(* Logix 5000 project; controller AdvManLab vendor 1 type 14 code 158 rev 28.12; software revision 28.01; part 2 of 13 *)
(* tags used below, declared in another part *)
   Inp : BOOL;   // Alarm Condition Input 1=Alarm
   Inp_Reset : BOOL;   // 1=Reset Alarm requiring reset
   Cfg_Exists : BOOL;   // 1=Alarm configured to exist, 0=Does not exist, don't scan
   Cfg_ResetReqd : BOOL;   // 1=Latched Alarm, a Reset is required to clear this Alarm
   Cfg_AckReqd : BOOL;   // 1=Acknowledge required for this Alarm
   Cfg_AllowShelve : BOOL;   // 1=Allow Operator to Shelve this Alarm
   Cfg_AllowDisable : BOOL;   // 1=Allow Maintenance to Disable this Alarm
   Cfg_PCmdClear : BOOL;   // 1=Clear Program Commands on receipt 0=Leave Set
   Cfg_Severity : INT;   // Alarm Severity: 1..250=Low, 251..500=Medium, 501..750=High, 751..1000=Urgent
   Cfg_AlmMinOnT : DINT;   // Minimum time Alm output stays on (sec)
   Cfg_MaxShelfT : INT;   // Auto unshelve after shelved this long (1..32767 minutes)
   PCfg_AllowExist : BOOL;   // 1=Alarm can be configured to exist, 0=other configs make alarm meaningless
   PCmd_Reset : BOOL;   // Program Command to Reset latched alarm
   PCmd_Ack : BOOL;   // Program Command to Acknowledge alarm
   PCmd_Suppress : BOOL;   // Program Command to Suppress by Design (inhibits new alarm)
   PCmd_Unsuppress : BOOL;   // Program Command to Unsuppress (allows new alarm)
   PCmd_Unshelve : BOOL;   // Program Command to Unshelve (e.g., on shift change)
   OCmd_Reset : BOOL;   // Operator Command to Reset latched alarm
   OCmd_Ack : BOOL;   // Operator Command to Acknowledge alarm
   OCmd_Shelve : BOOL;   // Operator Command to Shelve Alarm (inhibits new alarm)
   OCmd_Unshelve : BOOL;   // Operator Command to Unshelve alarm (allows new alarm)
   MCmd_Disable : BOOL;   // Maintenance Command to Disable alarm (inhibits new alarm)
   MCmd_Enable : BOOL;   // Maintenance Command to Enable alarm (allows new alarm)
   MCmd_Test : BOOL;   // Maintenance Command to Test alarm (issued for minimum alarm time)
   Val_Notify : SINT;   // Current Alarm Severity and Acknowledgement (enumeration)
   Val_MinToUnshelve : DINT;   // Number of minutes until this alarm unshelves itself (mmm:ss)
   Val_SecToUnshelve : DINT;   // Number of Seconds until this alarm unshelves itself (mmm:ss)
   Alm : ALIAS FOR Com_AE.0;   // Alarm output 1=In Alarm
   Ack : ALIAS FOR Com_AE.1;   // Alarm acknowledged status: 1=Ack rcvd
   Shelved : ALIAS FOR Com_AE.3;   // 1=Alarm has been Shelved by Operator (inhibits new alarm)
   Suppressed : ALIAS FOR Com_AE.6;   // 1=Alarm has been Suppressed by Program (inhibits new alarm)
   Disabled : ALIAS FOR Com_AE.9;   // 1=Alarm has been Disabled by Maintanance (inhibits new alarm)
   Sts_AlmInh : BOOL;   // 1=Alarm has been suppressed, shelved or disabled, display "I" icon
   Sts_Err : BOOL;   // 1=Error in Config: see detail Err_ bits for reason
   Err_Timer : BOOL;   // 1=Error in Config: Alarm Min On Time, Shelf Time (use 0 to 2147483)
   Err_Severity : BOOL;   // 1=Error in Config: Invalid Severity (use 1 to 4)
   Rdy_Reset : BOOL;   // Ready to receive OCmd_Reset (enables button)
   Rdy_Ack : BOOL;   // Ready to receive OCmd_Ack (enables button)
   Rdy_Shelve : BOOL;   // Ready to receive OCmd_Shelve (enables button)
   Rdy_Unshelve : BOOL;   // Ready to receive OCmd_Unshelve (enables button)
   Rdy_Disable : BOOL;   // Ready to receive MCmd_Disable (enables button)
   Rdy_Enable : BOOL;   // Ready to receive MCmd_Enable (enables button)
   Rdy_Test : BOOL;   // Ready to receive MCmd_Test (enables button)
   P_Alarm : BOOL;   // Unique Parameter Name for auto - discovery
   Wrk_Alm : BOOL;   // Internal Alarm Status
   Wrk_Suppressed : BOOL;   // Internal Alarm Suppressed Status
   Wrk_AlmMinOnT : TIMER;   // Alarm output minimum ON time to be seen by alarm server
   Wrk_AutoAckT : TIMER;   // Time to clear Ack bit when Ack not required
   Wrk_ShelfT : TIMER;   // Time to auto Unshelve a Shelved Alarm
   Com_AE : INT;   // Communication with HMI / Alarm/Event Server (see bit descriptions)
   Cfg_Tag : STRING_20;   // Alarm Tag Text (e.g., "LAHH-101")
   Cfg_Cond : STRING_20;   // Alarm Condition Text (e.g., "High-High PV")
   Wrk_SecToUnshelve : DINT;   // Number of seconds until this alarm unshelves itself
   Inf_Lib : STRING_12;   // Display Library for Faceplate call-up
   Inf_Type : STRING_16;   // Must contain AOI name, used for HMI and Information S/W
(* P_Alarm, continued *)

ROUTINE EnableInFalse   (* ladder *)
// Perform Alarm processing, but Invert Alarm Input ("Inp") for use on LD rung (EnableIn False)
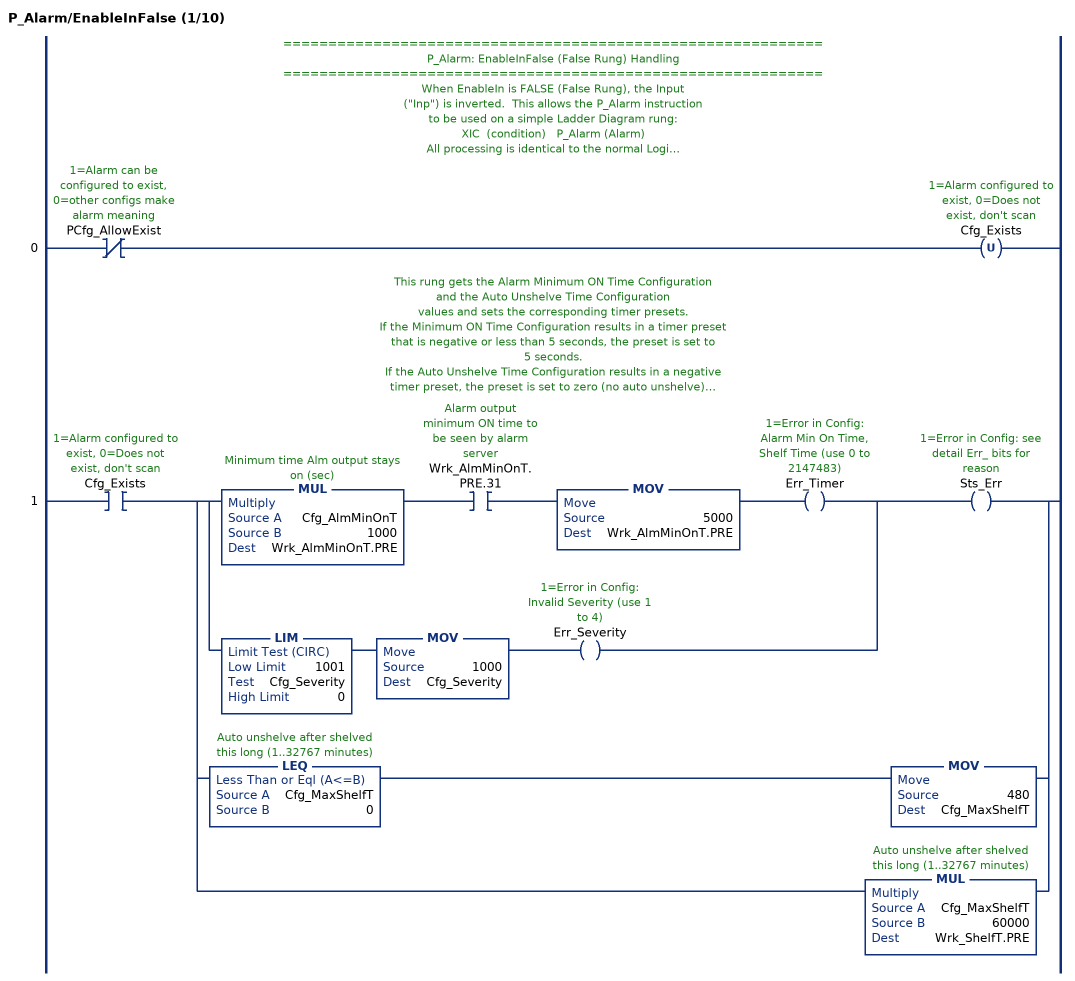
   // ============================================================
   // P_Alarm: EnableInFalse (False Rung) Handling
   // ============================================================
   // When EnableIn is FALSE (False Rung), the Input
   // ("Inp") is inverted.  This allows the P_Alarm instruction
   // to be used on a simple Ladder Diagram rung:
   // XIC  (condition)   P_Alarm (Alarm)
   // All processing is identical to the normal Logic
   // routine, except references to Inp are inverted!
   // ============================================================
   // CONFIGURATION
   // ============================================================
   // In the object containing this alarm, other configuration (such as not having
   // any limit switches) may make this particular alarm meaningless.
   // The Program Configuration "Allow Exist" is used to hide this alarm
   // on the object's faceplate and other graphics, and forces the Cfg_Exist to 0.
   // #####  V3.0-00  2013-06-30:  Added PCfg_AllowExist.  #####
   0: XIO(PCfg_AllowExist)OTU(Cfg_Exists);
   // This rung gets the Alarm Minimum ON Time Configuration
   // and the Auto Unshelve Time Configuration
   // values and sets the corresponding timer presets.
   // If the Minimum ON Time Configuration results in a timer preset
   // that is negative or less than 5 seconds, the preset is set to
   // 5 seconds.
   // If the Auto Unshelve Time Configuration results in a negative
   // timer preset, the preset is set to zero (no auto unshelve).
   //   The bad Config is flagged (Err_Timer).
   // Bad Config is also flagged if the Cfg_Severity is out of range (valid = 1..4)
   // #####  V3.0-00  2013-06-30:  Changed Program Inhibit to Suppress, Operator Suppress to Shelve.  #####
   // #####  Added Shelf Timer config check; if Severity out of range, make it "Fault".  #####
   // #####  V3.0-02  2013-10-30:  Changed Cfg_MaxShelfT check to LEQ 0.  (INT 1 to 32767 is valid.)  #####
   1: XIC(Cfg_Exists)[[MUL(Cfg_AlmMinOnT,1000,Wrk_AlmMinOnT.PRE) XIC(Wrk_AlmMinOnT.PRE.31) MOV(5000,Wrk_AlmMinOnT.PRE) OTE(Err_Timer) ,LIM(1001,Cfg_Severity,0) MOV(1000,Cfg_Severity) OTE(Err_Severity) ] OTE(Sts_Err) ,LEQ(Cfg_MaxShelfT,0) MOV(480,Cfg_MaxShelfT) ,MUL(Cfg_MaxShelfT,60000,Wrk_ShelfT.PRE) ];
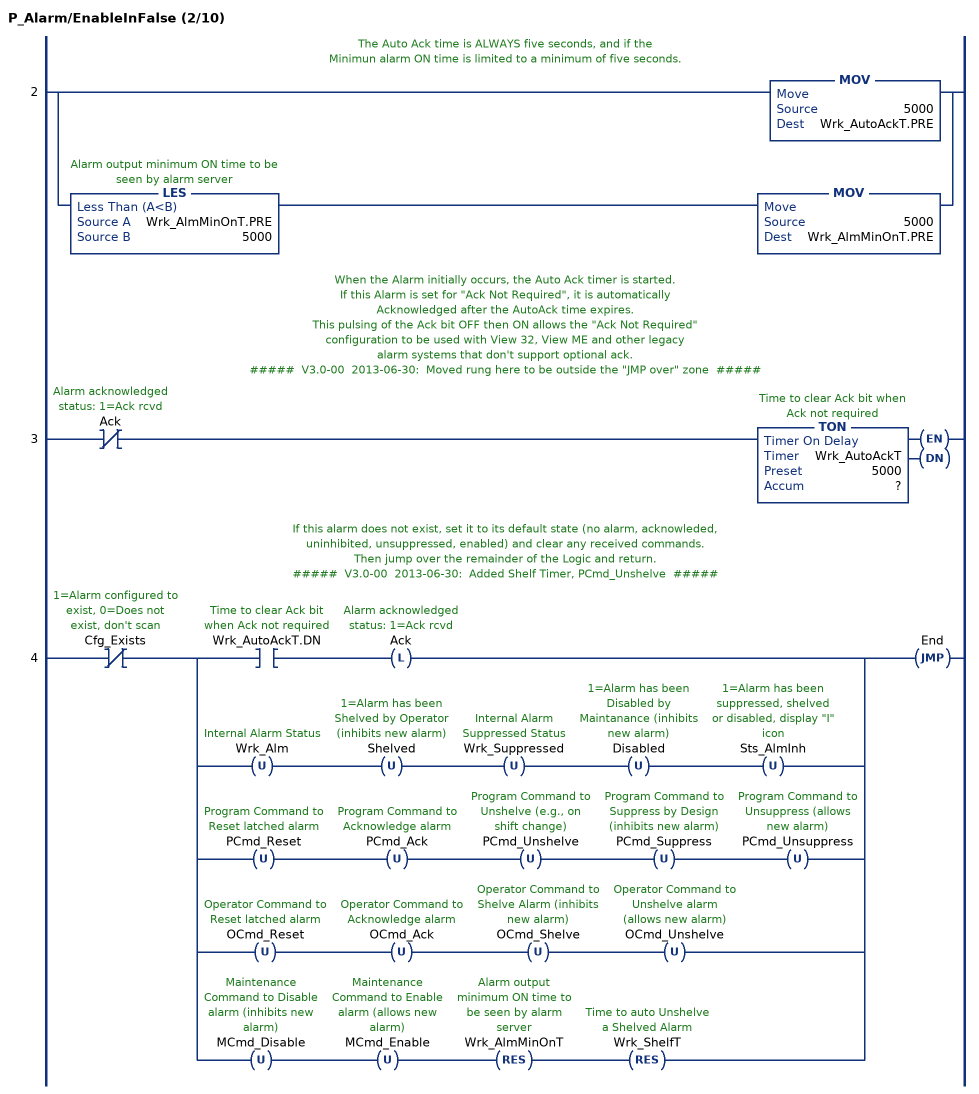
   // The Auto Ack time is ALWAYS five seconds, and if the
   // Minimun alarm ON time is limited to a minimum of five seconds.
   2: [MOV(5000,Wrk_AutoAckT.PRE) ,LES(Wrk_AlmMinOnT.PRE,5000) MOV(5000,Wrk_AlmMinOnT.PRE) ];
   // When the Alarm initially occurs, the Auto Ack timer is started.
   // If this Alarm is set for "Ack Not Required", it is automatically
   // Acknowledged after the AutoAck time expires.
   // This pulsing of the Ack bit OFF then ON allows the "Ack Not Required"
   // configuration to be used with View 32, View ME and other legacy
   // alarm systems that don't support optional ack.
   // #####  V3.0-00  2013-06-30:  Moved rung here to be outside the "JMP over" zone  #####
   3: XIO(Ack)TON(Wrk_AutoAckT,?,?);
   // If this alarm does not exist, set it to its default state (no alarm, acknowleded,
   // uninhibited, unsuppressed, enabled) and clear any received commands.
   // Then jump over the remainder of the Logic and return.
   // #####  V3.0-00  2013-06-30:  Added Shelf Timer, PCmd_Unshelve  #####
   4: XIO(Cfg_Exists)[XIC(Wrk_AutoAckT.DN) OTL(Ack) ,OTU(Wrk_Alm) OTU(Shelved) OTU(Wrk_Suppressed) OTU(Disabled) OTU(Sts_AlmInh) ,OTU(PCmd_Reset) OTU(PCmd_Ack) OTU(PCmd_Unshelve) OTU(PCmd_Suppress) OTU(PCmd_Unsuppress) ,OTU(OCmd_Reset) OTU(OCmd_Ack) OTU(OCmd_Shelve) OTU(OCmd_Unshelve) ,OTU(MCmd_Disable) OTU(MCmd_Enable) RES(Wrk_AlmMinOnT) RES(Wrk_ShelfT) ]JMP(End);
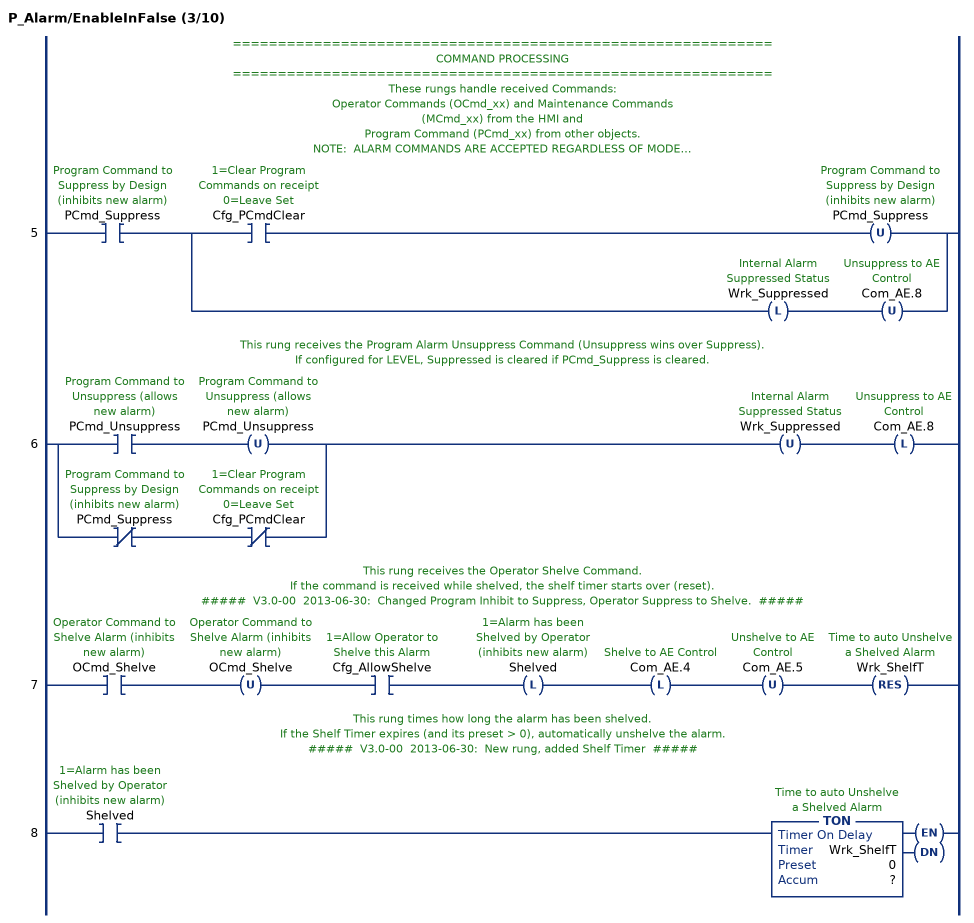
   // ============================================================
   // COMMAND PROCESSING
   // ============================================================
   // These rungs handle received Commands:
   // Operator Commands (OCmd_xx) and Maintenance Commands
   // (MCmd_xx) from the HMI and
   // Program Command (PCmd_xx) from other objects.
   // NOTE:  ALARM COMMANDS ARE ACCEPTED REGARDLESS OF MODE.
   // This rung receives the Program Alarm Inhibit Command.
   // If configured for EDGE, the Command is cleared.
   5: XIC(PCmd_Suppress)[XIC(Cfg_PCmdClear) OTU(PCmd_Suppress) ,OTL(Wrk_Suppressed) OTU(Com_AE.8) ];
   // This rung receives the Program Alarm Unsuppress Command (Unsuppress wins over Suppress).
   // If configured for LEVEL, Suppressed is cleared if PCmd_Suppress is cleared.
   6: [XIC(PCmd_Unsuppress) OTU(PCmd_Unsuppress) ,XIO(PCmd_Suppress) XIO(Cfg_PCmdClear) ]OTU(Wrk_Suppressed)OTL(Com_AE.8);
   // This rung receives the Operator Shelve Command.
   // If the command is received while shelved, the shelf timer starts over (reset).
   // #####  V3.0-00  2013-06-30:  Changed Program Inhibit to Suppress, Operator Suppress to Shelve.  #####
   7: XIC(OCmd_Shelve)OTU(OCmd_Shelve)XIC(Cfg_AllowShelve)OTL(Shelved)OTL(Com_AE.4)OTU(Com_AE.5)RES(Wrk_ShelfT);
   // This rung times how long the alarm has been shelved.
   // If the Shelf Timer expires (and its preset > 0), automatically unshelve the alarm.
   // #####  V3.0-00  2013-06-30:  New rung, added Shelf Timer  #####
   8: XIC(Shelved)TON(Wrk_ShelfT,?,?);
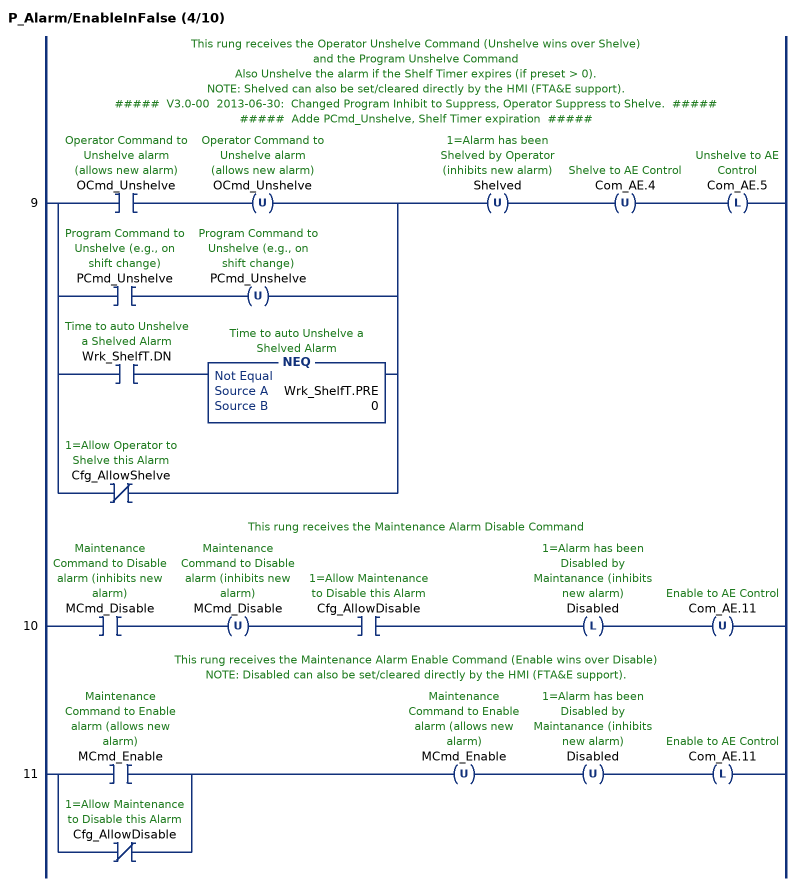
   // This rung receives the Operator Unshelve Command (Unshelve wins over Shelve)
   // and the Program Unshelve Command
   // Also Unshelve the alarm if the Shelf Timer expires (if preset > 0).
   // NOTE: Shelved can also be set/cleared directly by the HMI (FTA&E support).
   // #####  V3.0-00  2013-06-30:  Changed Program Inhibit to Suppress, Operator Suppress to Shelve.  #####
   // #####  Adde PCmd_Unshelve, Shelf Timer expiration  #####
   9: [XIC(OCmd_Unshelve) OTU(OCmd_Unshelve) ,XIC(PCmd_Unshelve) OTU(PCmd_Unshelve) ,XIC(Wrk_ShelfT.DN) NEQ(Wrk_ShelfT.PRE,0) ,XIO(Cfg_AllowShelve) ]OTU(Shelved)OTU(Com_AE.4)OTL(Com_AE.5);
   // This rung receives the Maintenance Alarm Disable Command
   10: XIC(MCmd_Disable)OTU(MCmd_Disable)XIC(Cfg_AllowDisable)OTL(Disabled)OTU(Com_AE.11);
   // This rung receives the Maintenance Alarm Enable Command (Enable wins over Disable)
   // NOTE: Disabled can also be set/cleared directly by the HMI (FTA&E support).
   11: [XIC(MCmd_Enable) ,XIO(Cfg_AllowDisable) ]OTU(MCmd_Enable)OTU(Disabled)OTL(Com_AE.11);
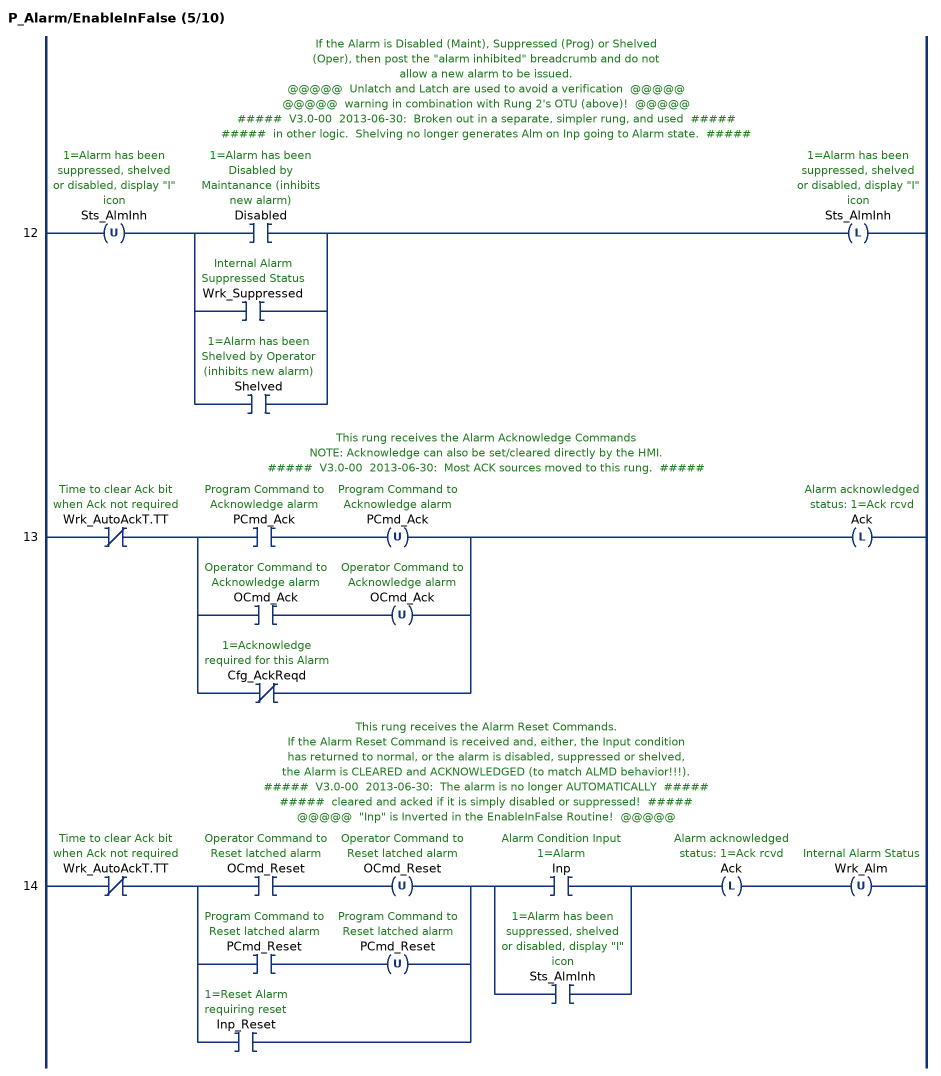
   // If the Alarm is Disabled (Maint), Suppressed (Prog) or Shelved
   // (Oper), then post the "alarm inhibited" breadcrumb and do not
   // allow a new alarm to be issued.
   // @@@@@  Unlatch and Latch are used to avoid a verification  @@@@@
   // @@@@@  warning in combination with Rung 2's OTU (above)!  @@@@@
   // #####  V3.0-00  2013-06-30:  Broken out in a separate, simpler rung, and used  #####
   // #####  in other logic.  Shelving no longer generates Alm on Inp going to Alarm state.  #####
   12: OTU(Sts_AlmInh)[XIC(Disabled) ,XIC(Wrk_Suppressed) ,XIC(Shelved) ]OTL(Sts_AlmInh);
   // This rung receives the Alarm Acknowledge Commands
   // NOTE: Acknowledge can also be set/cleared directly by the HMI.
   // #####  V3.0-00  2013-06-30:  Most ACK sources moved to this rung.  #####
   13: XIO(Wrk_AutoAckT.TT)[XIC(PCmd_Ack) OTU(PCmd_Ack) ,XIC(OCmd_Ack) OTU(OCmd_Ack) ,XIO(Cfg_AckReqd) ]OTL(Ack);
   // This rung receives the Alarm Reset Commands.
   // If the Alarm Reset Command is received and, either, the Input condition
   // has returned to normal, or the alarm is disabled, suppressed or shelved,
   // the Alarm is CLEARED and ACKNOWLEDGED (to match ALMD behavior!!!).
   // #####  V3.0-00  2013-06-30:  The alarm is no longer AUTOMATICALLY  #####
   // #####  cleared and acked if it is simply disabled or suppressed!  #####
   // @@@@@  "Inp" is Inverted in the EnableInFalse Routine!  @@@@@
   14: XIO(Wrk_AutoAckT.TT)[XIC(OCmd_Reset) OTU(OCmd_Reset) ,XIC(PCmd_Reset) OTU(PCmd_Reset) ,XIC(Inp_Reset) ][XIC(Inp) ,XIC(Sts_AlmInh) ]OTL(Ack)OTU(Wrk_Alm);
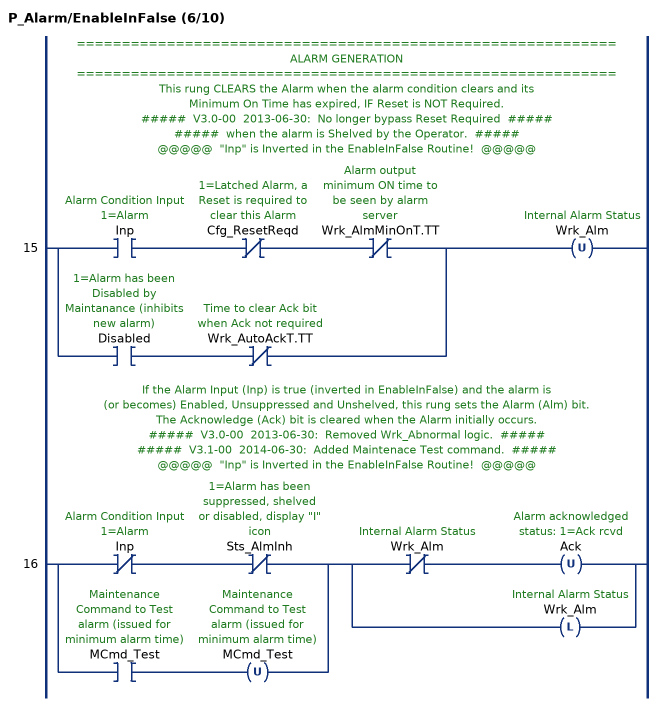
   // ============================================================
   // ALARM GENERATION
   // ============================================================
   // This rung CLEARS the Alarm when the alarm condition clears and its
   // Minimum On Time has expired, IF Reset is NOT Required.
   // #####  V3.0-00  2013-06-30:  No longer bypass Reset Required  #####
   // #####  when the alarm is Shelved by the Operator.  #####
   // @@@@@  "Inp" is Inverted in the EnableInFalse Routine!  @@@@@
   15: [XIC(Inp) XIO(Cfg_ResetReqd) XIO(Wrk_AlmMinOnT.TT) ,XIC(Disabled) XIO(Wrk_AutoAckT.TT) ]OTU(Wrk_Alm);
   // If the Alarm Input (Inp) is true (inverted in EnableInFalse) and the alarm is
   // (or becomes) Enabled, Unsuppressed and Unshelved, this rung sets the Alarm (Alm) bit.
   // The Acknowledge (Ack) bit is cleared when the Alarm initially occurs.
   // #####  V3.0-00  2013-06-30:  Removed Wrk_Abnormal logic.  #####
   // #####  V3.1-00  2014-06-30:  Added Maintenace Test command.  #####
   // @@@@@  "Inp" is Inverted in the EnableInFalse Routine!  @@@@@
   16: [XIO(Inp) XIO(Sts_AlmInh) ,XIC(MCmd_Test) OTU(MCmd_Test) ][XIO(Wrk_Alm) OTU(Ack) ,OTL(Wrk_Alm) ];
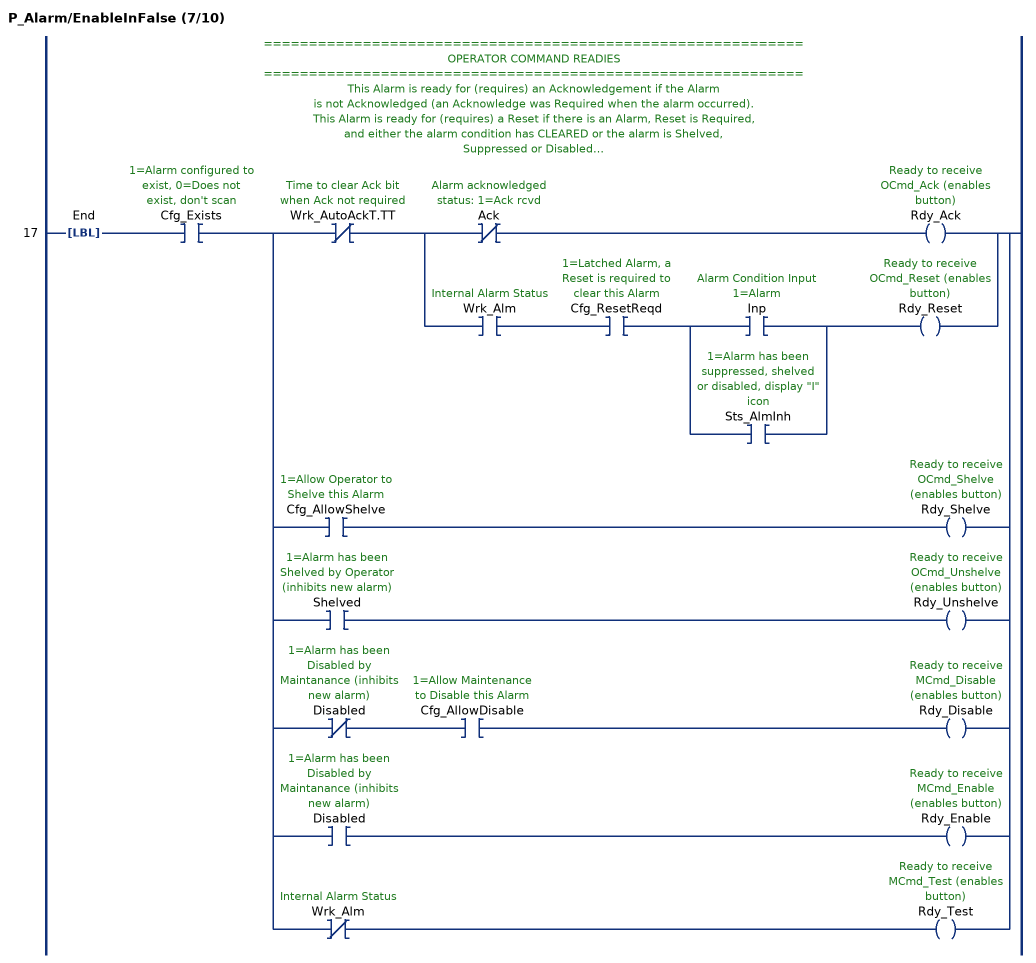
   // ============================================================
   // OPERATOR COMMAND READIES
   // ============================================================
   // This Alarm is ready for (requires) an Acknowledgement if the Alarm
   // is not Acknowledged (an Acknowledge was Required when the alarm occurred).
   // This Alarm is ready for (requires) a Reset if there is an Alarm, Reset is Required,
   // and either the alarm condition has CLEARED or the alarm is Shelved,
   // Suppressed or Disabled.
   // .
   // If the Alarm is NOT Shelved, it is ready for Shelve.
   // If the Alarm IS Shelved, it is ready for Unshelve.
   // If the Alarm is NOT Disabled, it is ready for Disable.
   // If the Alarm IS Disabled, it is ready for Enable.
   // NOTE: This rung appears before the Values/Status rung because the Rdy_Reset
   // condition is used to eliminate redundant logic in the rung below for Val_Notify.0.
   // #####  V3.0-00  2013-06-30:  Added sub-branch with Sts_AlmInh  #####
   // #####  V3.1-00  2014-06-30:  Added Maintenace Test command.  #####
   // @@@@@  "Inp" is Inverted in the EnableInFalse Routine!  @@@@@
   17: LBL(End)XIC(Cfg_Exists)[XIO(Wrk_AutoAckT.TT) [XIO(Ack) OTE(Rdy_Ack) ,XIC(Wrk_Alm) XIC(Cfg_ResetReqd) [XIC(Inp) ,XIC(Sts_AlmInh) ] OTE(Rdy_Reset) ] ,XIC(Cfg_AllowShelve) OTE(Rdy_Shelve) ,XIC(Shelved) OTE(Rdy_Unshelve) ,XIO(Disabled) XIC(Cfg_AllowDisable) OTE(Rdy_Disable) ,XIC(Disabled) OTE(Rdy_Enable) ,XIO(Wrk_Alm) OTE(Rdy_Test) ];
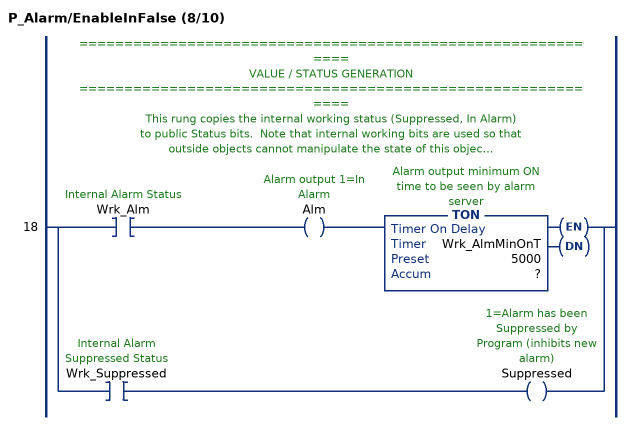
   // ============================================================
   // VALUE / STATUS GENERATION
   // ============================================================
   // This rung copies the internal working status (Suppressed, In Alarm)
   // to public Status bits.  Note that internal working bits are used so that
   // outside objects cannot manipulate the state of this object
   // by setting/clearing its Status and Alarm bits.
   // Public Status is generated for:
   // Alarm (with minimum ON time to be seen by polling)
   // Alarm Suppressed
   // Unsuppressed, Unshelved and Enabled are generated for HMI (FTVSE 7).
   // (Ack, Shelved and Disabled can be set/cleared by the HMI directly.
   // Note that these bits are "read/write" outputs in the parameter definition.)
   // #####  V3.0-00  2013-06-30:  New rung, some from below, new HMI bits.  #####
   18: [XIC(Wrk_Alm) OTE(Alm) TON(Wrk_AlmMinOnT,?,?) ,XIC(Wrk_Suppressed) OTE(Suppressed) ];
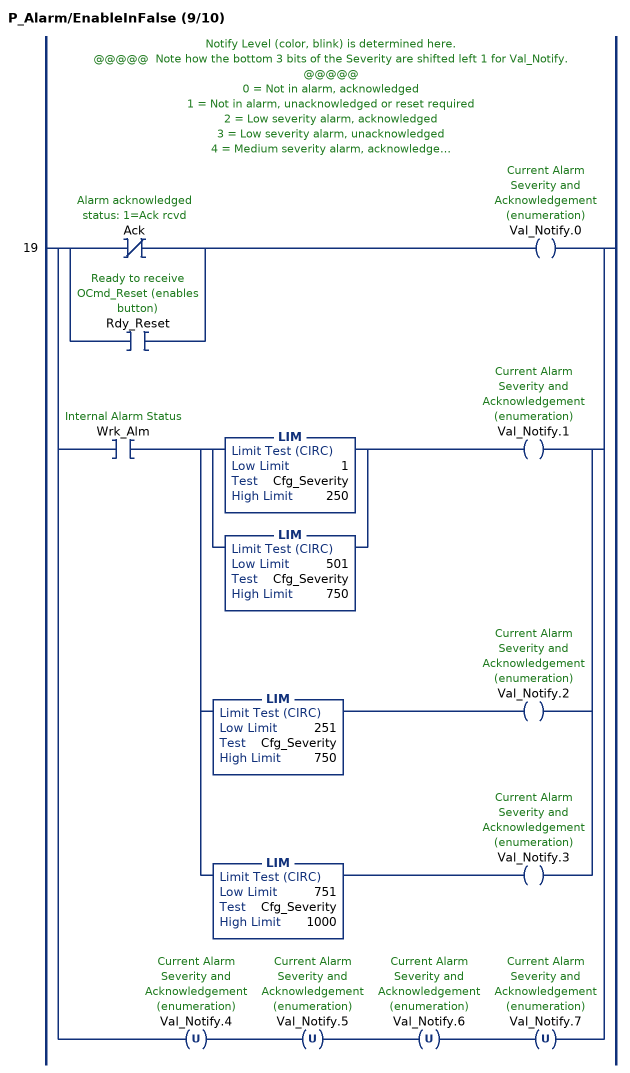
   // Notify Level (color, blink) is determined here.
   // @@@@@  Note how the bottom 3 bits of the Severity are shifted left 1 for Val_Notify.  @@@@@
   // 0 = Not in alarm, acknowledged
   // 1 = Not in alarm, unacknowledged or reset required
   // 2 = Low severity alarm, acknowledged
   // 3 = Low severity alarm, unacknowledged
   // 4 = Medium severity alarm, acknowledged
   // 5 = Medium severity alarm, unacknowledged
   // 6 = High severity alarm, acknowledged
   // 7 = High severity alarm, unacknowledged
   // 8 = Urgent severity alarm, acknowledged
   // 9 = Urgent severity alarm, unacknowledged
   // NOTE that the alarm bell icon will blink, even though the alarm is Acknowledged,
   // if an Alarm Reset is required (to get the Operator's attention).
   // #####  V3.0-00  2013-06-30:  Moved a few functions off this rung to logic above.  #####
   // #####  Names of Severity levels changed to Low, Medium, High, Highest  #####
   // #####  to match examples in ANSI/ISA-18.2-2009.  #####
   // #####  V3.1-00  2014-06-30:  Changed severity ranges, names to match FTAE  #####
   19: [[XIO(Ack) ,XIC(Rdy_Reset) ] OTE(Val_Notify.0) ,XIC(Wrk_Alm) [[LIM(1,Cfg_Severity,250) ,LIM(501,Cfg_Severity,750) ] OTE(Val_Notify.1) ,LIM(251,Cfg_Severity,750) OTE(Val_Notify.2) ,LIM(751,Cfg_Severity,1000) OTE(Val_Notify.3) ] ,OTU(Val_Notify.4) OTU(Val_Notify.5) OTU(Val_Notify.6) OTU(Val_Notify.7) ];
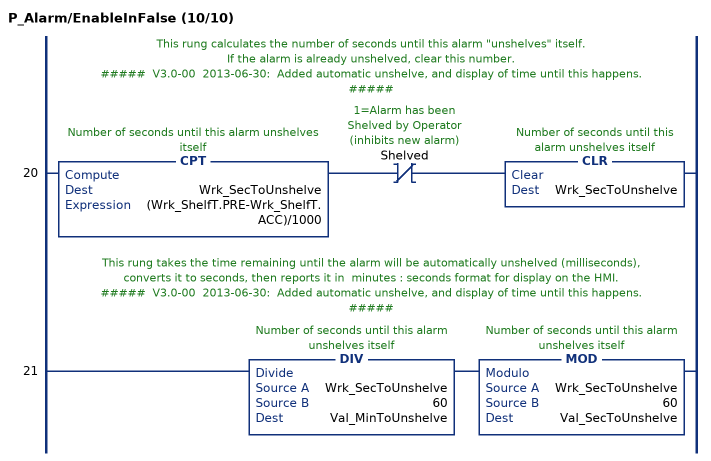
   // This rung calculates the number of seconds until this alarm "unshelves" itself.
   // If the alarm is already unshelved, clear this number.
   // #####  V3.0-00  2013-06-30:  Added automatic unshelve, and display of time until this happens.  #####
   20: CPT(Wrk_SecToUnshelve,(Wrk_ShelfT.PRE-Wrk_ShelfT.ACC)/1000)XIO(Shelved)CLR(Wrk_SecToUnshelve);
   // This rung takes the time remaining until the alarm will be automatically unshelved (milliseconds),
   // converts it to seconds, then reports it in  minutes : seconds format for display on the HMI.
   // #####  V3.0-00  2013-06-30:  Added automatic unshelve, and display of time until this happens.  #####
   21: DIV(Wrk_SecToUnshelve,60,Val_MinToUnshelve)MOD(Wrk_SecToUnshelve,60,Val_SecToUnshelve);
END_ROUTINE

ROUTINE Logic   (* ladder *)
// Perform Alarm processing: delay, latch/reset, acknowledge, enable/disable, inhibit/uninhibit, suppress/unsuppress
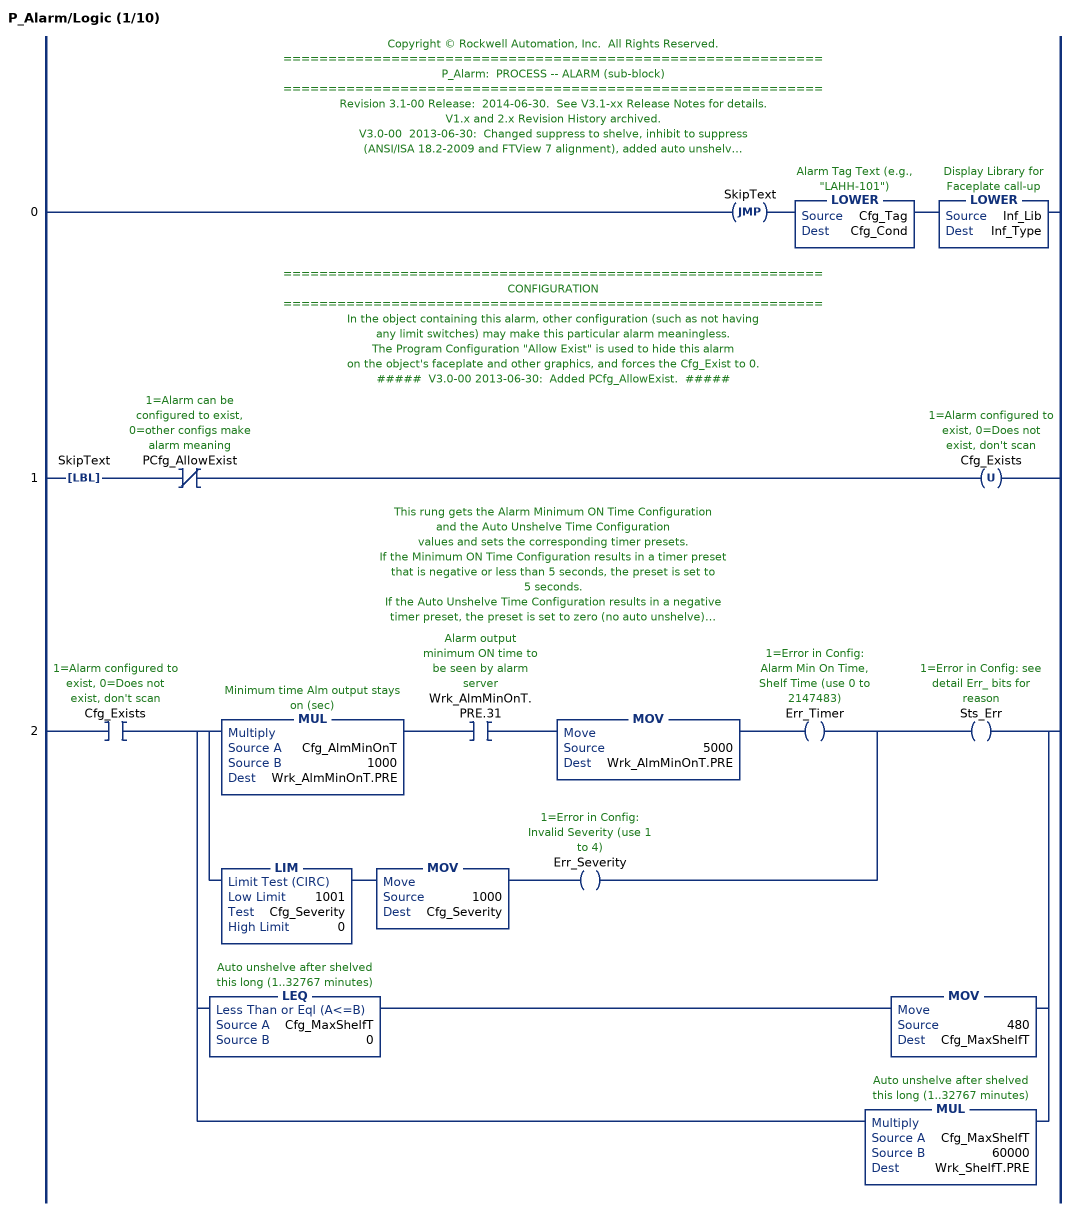
   // Copyright © Rockwell Automation, Inc.  All Rights Reserved.
   // ============================================================
   // P_Alarm:  PROCESS -- ALARM (sub-block)
   // ============================================================
   // Revision 3.1-00 Release:  2014-06-30.  See V3.1-xx Release Notes for details.
   // V1.x and 2.x Revision History archived.
   // V3.0-00  2013-06-30:  Changed suppress to shelve, inhibit to suppress
   // (ANSI/ISA 18.2-2009 and FTView 7 alignment), added auto unshelve
   // timer, program command to unshelve.  Removed: Ack on shelve.
   // Added: clear Alm when Disabled, PCfg_AllowExist, Cfg_Tag,
   // Cfg_Cond, Inf_Lib, Inf_Type.  (Max Shelf Time is in MINUTES.)
   // Added local tag .Com_AE for FTAE communications.
   // V3.0-01  2013-07-30:  Changed range for Shelf Time to 1 to 34560 minutes.
   // V3.0-02  2013-10-30:  Changed Cfg_MaxShelfT check to LEQ 0.
   // (INT 1 to 32767 is valid.)
   // V3.1-00  2014-06-30:  Added Maintenace Test command, changed severity
   // ranges and names to match FTAE (for linking to FTView 8).
   // ============================================================
   // This instruction monitors one input condition and provides one Alarm with:
   //   * configurable latching (reset required) and acknowledgement requirement
   //   * configurable alarm severity
   // 1..250 = Low  (blue, typ. informational)
   // 251-500 = Medium  (yelllow, typ. warning)
   // 501-750 = High  (red, typ. process exception)
   // 751-1000 = Urgent  (magenta, typ. equip. fault)
   // * configurable minimum ON time (e.g., to ensure it is seen by the HMI)
   // * commands to suppress/unsuppress (Prog), shelve/unshelve (Oper)
   // and disable/enable (Maint) the alarm.
   // * configurable amount of time shelved to automatically unshelve an alarm
   // * FTA&E support for suppressed, shelved and disabled states (V7.0)
   // NOTE regarding parameter naming:
   // FTA&E names (same as ALMD instruction) are used instead
   // of the ANSI/ISA 18.2-2009 names, as follows:
   // "Disabled" is the equivalent of "Out of Service" in ISA 18.2.
   // (the Disabled state is owned by Maintenance)
   // "Suppressed" is the equivalent of "Suppressed by Design" in ISA 18.2.
   // (the Suppressed state is owned by Program logic)
   // "Shelved" is the same as in ISA 18.2.
   // (the Shelved state is owned by Operator, but may be cleared
   // by Program logic based on time, shift change, etc.)
   // This instruction is usually nested within other instructions, with one instance
   // used for each Alarm generated by the containing instruction.  It may also be
   // used as a standalone instruction for Alarm conditions generated by custom logic.
   // ________________________________________
   // FTAE Alarm Setup:
   // ________________________________________
   // (object).(alarm).Com_AE.0:  Alarm to FTAE
   //     .Com_AE.1:   Ack to/from FTAE
   //     .Com_AE.3:   Shelved from FTAE Status
   //     .Com_AE.4:   Shelve/Reshelve to FTAE Control (auto reset)
   //     .Com_AE.5:   Unshelve to FTAE Control (auto reset)
   //     .Com_AE.6:   Suppressed to/from FTAE
   //     .Com_AE.8:   Unsuppress to FTAE Control (auto reset)
   //     .Com_AE.9:   Disabled to/from FTAE
   //     .Com_AE.11: Enable to FTAE Control (auto reset)
   // all other bits unused
   //     .Cfg_MaxShelfT is also used in FTAE config.
   // ============================================================
   // POWERUP / INVALID STATE HANDLING
   // ============================================================
   // All internal Work (state) bits maintain states through a power cycle and are
   // independent.  No first-scan logic is required.  See the Prescan routine for
   // powerup / prescan code.
   // ============================================================
   // SHOW LOCAL STRINGS
   // ============================================================
   // The STRINGs containing the text associated with each instance of this
   // instruction cannot be Input or Output Parameters, because STRINGs are not
   //  'atomic' types. (Inputs and Outputs must be SINT, INT, DINT, REAL, or BOOL.)
   // In order to make it easier to find and configure these STRINGs, this rung
   // was added.  THE JMP (and the LBL on the following rung)
   // MUST NOT BE REMOVED!!!
   // To view the STRINGs, go to the instruction instance (in LD or FBD), RIGHT-click
   // to bring up the context menu and select "Open Instruction Logic".
   // This rung will appear with the STRING values for the selected instance.
   // You may double-click the STRING values here to modify them as well.
   // #####  V3.0-00  2013-06-30:  Added rung; added new STRING local tags.  #####
   0: JMP(SkipText)LOWER(Cfg_Tag,Cfg_Cond)LOWER(Inf_Lib,Inf_Type);
   // ============================================================
   // CONFIGURATION
   // ============================================================
   // In the object containing this alarm, other configuration (such as not having
   // any limit switches) may make this particular alarm meaningless.
   // The Program Configuration "Allow Exist" is used to hide this alarm
   // on the object's faceplate and other graphics, and forces the Cfg_Exist to 0.
   // #####  V3.0-00 2013-06-30:  Added PCfg_AllowExist.  #####
   1: LBL(SkipText)XIO(PCfg_AllowExist)OTU(Cfg_Exists);
   // This rung gets the Alarm Minimum ON Time Configuration
   // and the Auto Unshelve Time Configuration
   // values and sets the corresponding timer presets.
   // If the Minimum ON Time Configuration results in a timer preset
   // that is negative or less than 5 seconds, the preset is set to
   // 5 seconds.
   // If the Auto Unshelve Time Configuration results in a negative
   // timer preset, the preset is set to zero (no auto unshelve).
   //   The bad Config is flagged (Err_Timer).
   // Bad Config is also flagged if the Cfg_Severity is out of range (valid = 1..4)
   // #####  V3.0-00  2013-06-30:  Changed Program Inhibit to Suppress, Operator Suppress to Shelve.  #####
   // #####  Added Shelf Timer config check; if Severity out of range, make it "Fault".  #####
   // #####  V3.0-02  2013-10-30:  Changed Cfg_MaxShelfT check to LEQ 0.  (INT 1 to 32767 is valid.)  #####
   2: XIC(Cfg_Exists)[[MUL(Cfg_AlmMinOnT,1000,Wrk_AlmMinOnT.PRE) XIC(Wrk_AlmMinOnT.PRE.31) MOV(5000,Wrk_AlmMinOnT.PRE) OTE(Err_Timer) ,LIM(1001,Cfg_Severity,0) MOV(1000,Cfg_Severity) OTE(Err_Severity) ] OTE(Sts_Err) ,LEQ(Cfg_MaxShelfT,0) MOV(480,Cfg_MaxShelfT) ,MUL(Cfg_MaxShelfT,60000,Wrk_ShelfT.PRE) ];
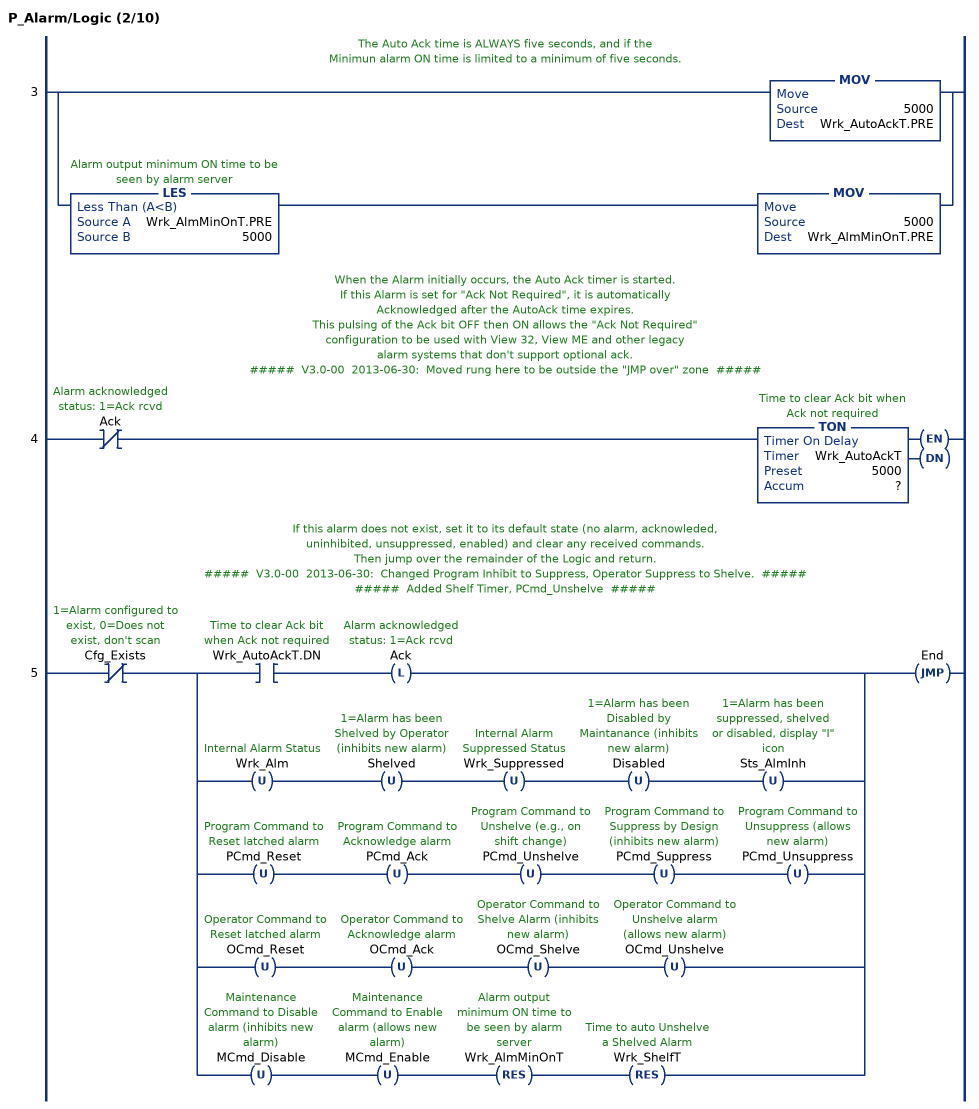
   // The Auto Ack time is ALWAYS five seconds, and if the
   // Minimun alarm ON time is limited to a minimum of five seconds.
   3: [MOV(5000,Wrk_AutoAckT.PRE) ,LES(Wrk_AlmMinOnT.PRE,5000) MOV(5000,Wrk_AlmMinOnT.PRE) ];
   // When the Alarm initially occurs, the Auto Ack timer is started.
   // If this Alarm is set for "Ack Not Required", it is automatically
   // Acknowledged after the AutoAck time expires.
   // This pulsing of the Ack bit OFF then ON allows the "Ack Not Required"
   // configuration to be used with View 32, View ME and other legacy
   // alarm systems that don't support optional ack.
   // #####  V3.0-00  2013-06-30:  Moved rung here to be outside the "JMP over" zone  #####
   4: XIO(Ack)TON(Wrk_AutoAckT,?,?);
   // If this alarm does not exist, set it to its default state (no alarm, acknowleded,
   // uninhibited, unsuppressed, enabled) and clear any received commands.
   // Then jump over the remainder of the Logic and return.
   // #####  V3.0-00  2013-06-30:  Changed Program Inhibit to Suppress, Operator Suppress to Shelve.  #####
   // #####  Added Shelf Timer, PCmd_Unshelve  #####
   5: XIO(Cfg_Exists)[XIC(Wrk_AutoAckT.DN) OTL(Ack) ,OTU(Wrk_Alm) OTU(Shelved) OTU(Wrk_Suppressed) OTU(Disabled) OTU(Sts_AlmInh) ,OTU(PCmd_Reset) OTU(PCmd_Ack) OTU(PCmd_Unshelve) OTU(PCmd_Suppress) OTU(PCmd_Unsuppress) ,OTU(OCmd_Reset) OTU(OCmd_Ack) OTU(OCmd_Shelve) OTU(OCmd_Unshelve) ,OTU(MCmd_Disable) OTU(MCmd_Enable) RES(Wrk_AlmMinOnT) RES(Wrk_ShelfT) ]JMP(End);
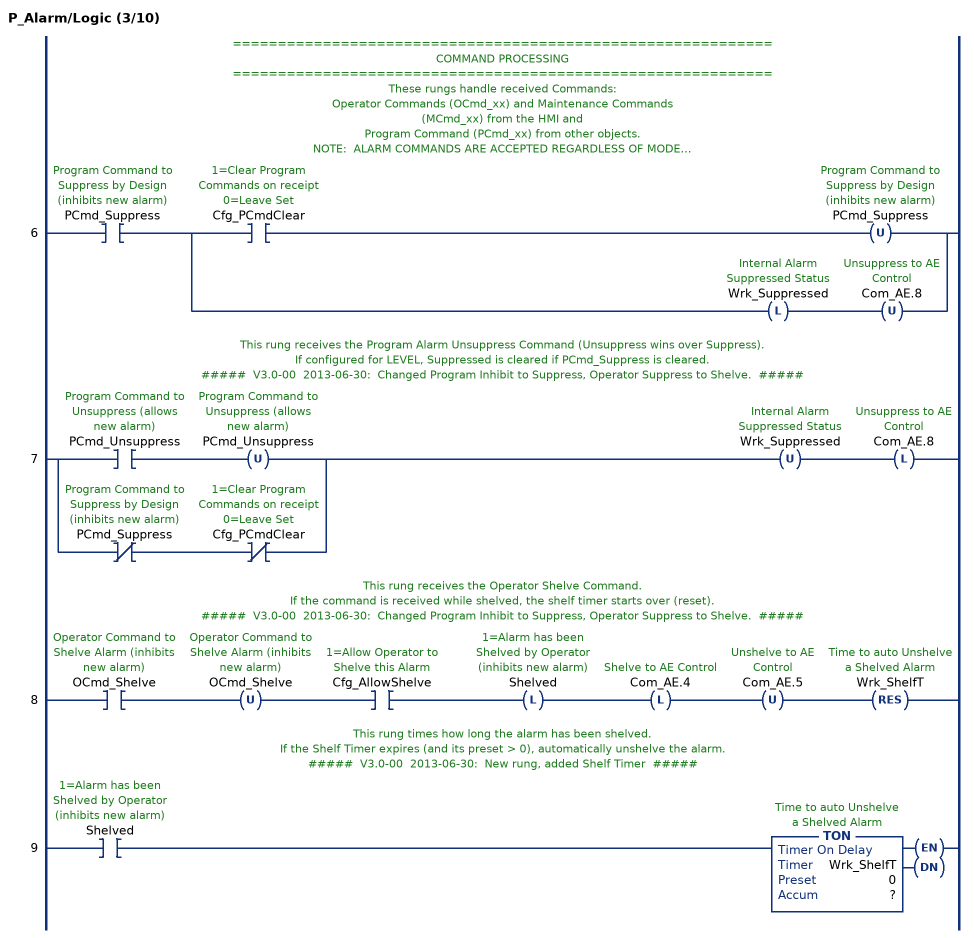
   // ============================================================
   // COMMAND PROCESSING
   // ============================================================
   // These rungs handle received Commands:
   // Operator Commands (OCmd_xx) and Maintenance Commands
   // (MCmd_xx) from the HMI and
   // Program Command (PCmd_xx) from other objects.
   // NOTE:  ALARM COMMANDS ARE ACCEPTED REGARDLESS OF MODE.
   // This rung receives the Program Alarm Inhibit Command.
   // If configured for EDGE, the Command is cleared.
   6: XIC(PCmd_Suppress)[XIC(Cfg_PCmdClear) OTU(PCmd_Suppress) ,OTL(Wrk_Suppressed) OTU(Com_AE.8) ];
   // This rung receives the Program Alarm Unsuppress Command (Unsuppress wins over Suppress).
   // If configured for LEVEL, Suppressed is cleared if PCmd_Suppress is cleared.
   // #####  V3.0-00  2013-06-30:  Changed Program Inhibit to Suppress, Operator Suppress to Shelve.  #####
   7: [XIC(PCmd_Unsuppress) OTU(PCmd_Unsuppress) ,XIO(PCmd_Suppress) XIO(Cfg_PCmdClear) ]OTU(Wrk_Suppressed)OTL(Com_AE.8);
   // This rung receives the Operator Shelve Command.
   // If the command is received while shelved, the shelf timer starts over (reset).
   // #####  V3.0-00  2013-06-30:  Changed Program Inhibit to Suppress, Operator Suppress to Shelve.  #####
   8: XIC(OCmd_Shelve)OTU(OCmd_Shelve)XIC(Cfg_AllowShelve)OTL(Shelved)OTL(Com_AE.4)OTU(Com_AE.5)RES(Wrk_ShelfT);
   // This rung times how long the alarm has been shelved.
   // If the Shelf Timer expires (and its preset > 0), automatically unshelve the alarm.
   // #####  V3.0-00  2013-06-30:  New rung, added Shelf Timer  #####
   9: XIC(Shelved)TON(Wrk_ShelfT,?,?);
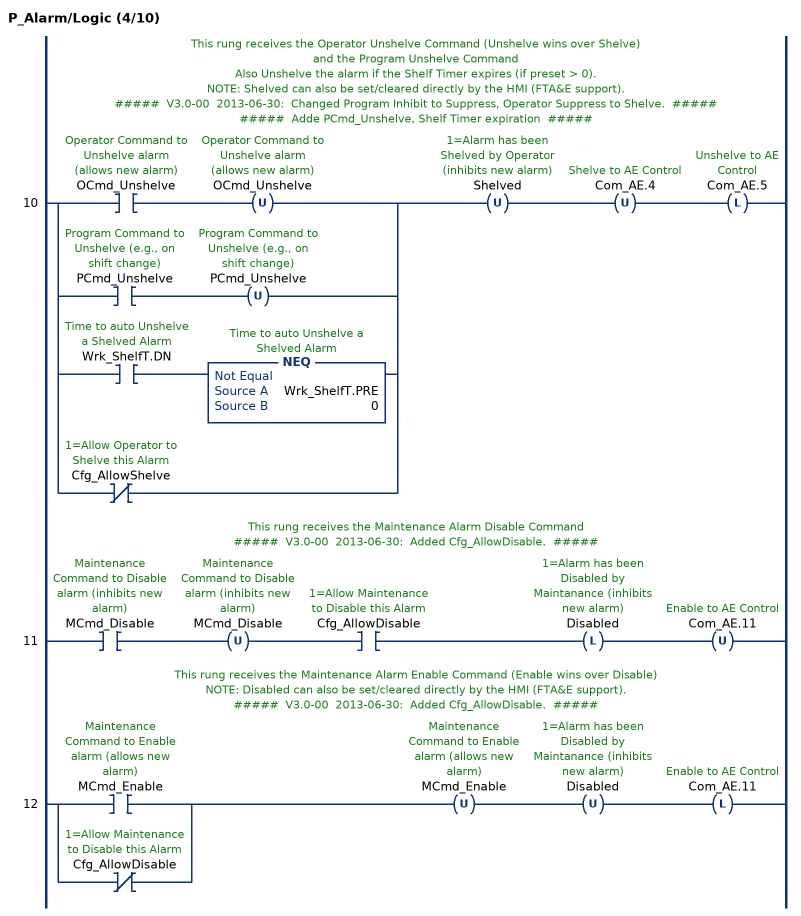
   // This rung receives the Operator Unshelve Command (Unshelve wins over Shelve)
   // and the Program Unshelve Command
   // Also Unshelve the alarm if the Shelf Timer expires (if preset > 0).
   // NOTE: Shelved can also be set/cleared directly by the HMI (FTA&E support).
   // #####  V3.0-00  2013-06-30:  Changed Program Inhibit to Suppress, Operator Suppress to Shelve.  #####
   // #####  Adde PCmd_Unshelve, Shelf Timer expiration  #####
   10: [XIC(OCmd_Unshelve) OTU(OCmd_Unshelve) ,XIC(PCmd_Unshelve) OTU(PCmd_Unshelve) ,XIC(Wrk_ShelfT.DN) NEQ(Wrk_ShelfT.PRE,0) ,XIO(Cfg_AllowShelve) ]OTU(Shelved)OTU(Com_AE.4)OTL(Com_AE.5);
   // This rung receives the Maintenance Alarm Disable Command
   // #####  V3.0-00  2013-06-30:  Added Cfg_AllowDisable.  #####
   11: XIC(MCmd_Disable)OTU(MCmd_Disable)XIC(Cfg_AllowDisable)OTL(Disabled)OTU(Com_AE.11);
   // This rung receives the Maintenance Alarm Enable Command (Enable wins over Disable)
   // NOTE: Disabled can also be set/cleared directly by the HMI (FTA&E support).
   // #####  V3.0-00  2013-06-30:  Added Cfg_AllowDisable.  #####
   12: [XIC(MCmd_Enable) ,XIO(Cfg_AllowDisable) ]OTU(MCmd_Enable)OTU(Disabled)OTL(Com_AE.11);
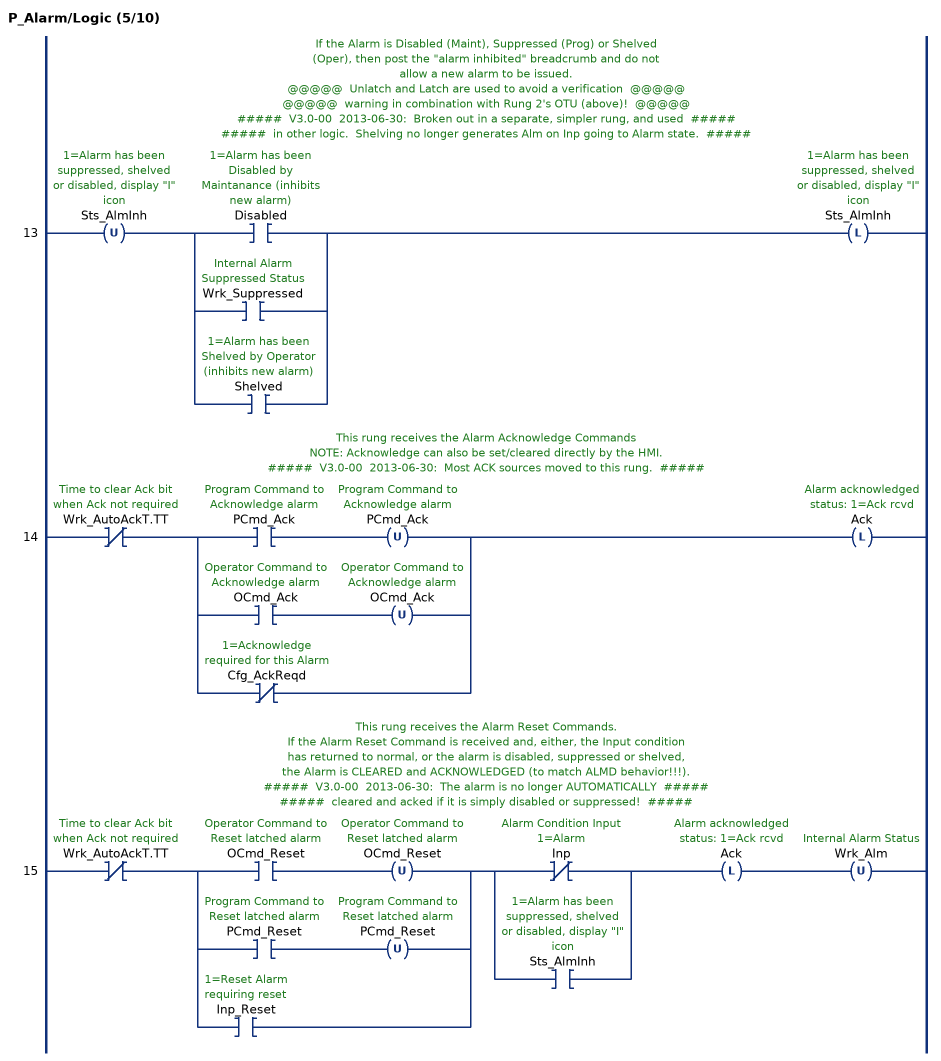
   // If the Alarm is Disabled (Maint), Suppressed (Prog) or Shelved
   // (Oper), then post the "alarm inhibited" breadcrumb and do not
   // allow a new alarm to be issued.
   // @@@@@  Unlatch and Latch are used to avoid a verification  @@@@@
   // @@@@@  warning in combination with Rung 2's OTU (above)!  @@@@@
   // #####  V3.0-00  2013-06-30:  Broken out in a separate, simpler rung, and used  #####
   // #####  in other logic.  Shelving no longer generates Alm on Inp going to Alarm state.  #####
   13: OTU(Sts_AlmInh)[XIC(Disabled) ,XIC(Wrk_Suppressed) ,XIC(Shelved) ]OTL(Sts_AlmInh);
   // This rung receives the Alarm Acknowledge Commands
   // NOTE: Acknowledge can also be set/cleared directly by the HMI.
   // #####  V3.0-00  2013-06-30:  Most ACK sources moved to this rung.  #####
   14: XIO(Wrk_AutoAckT.TT)[XIC(PCmd_Ack) OTU(PCmd_Ack) ,XIC(OCmd_Ack) OTU(OCmd_Ack) ,XIO(Cfg_AckReqd) ]OTL(Ack);
   // This rung receives the Alarm Reset Commands.
   // If the Alarm Reset Command is received and, either, the Input condition
   // has returned to normal, or the alarm is disabled, suppressed or shelved,
   // the Alarm is CLEARED and ACKNOWLEDGED (to match ALMD behavior!!!).
   // #####  V3.0-00  2013-06-30:  The alarm is no longer AUTOMATICALLY  #####
   // #####  cleared and acked if it is simply disabled or suppressed!  #####
   15: XIO(Wrk_AutoAckT.TT)[XIC(OCmd_Reset) OTU(OCmd_Reset) ,XIC(PCmd_Reset) OTU(PCmd_Reset) ,XIC(Inp_Reset) ][XIO(Inp) ,XIC(Sts_AlmInh) ]OTL(Ack)OTU(Wrk_Alm);
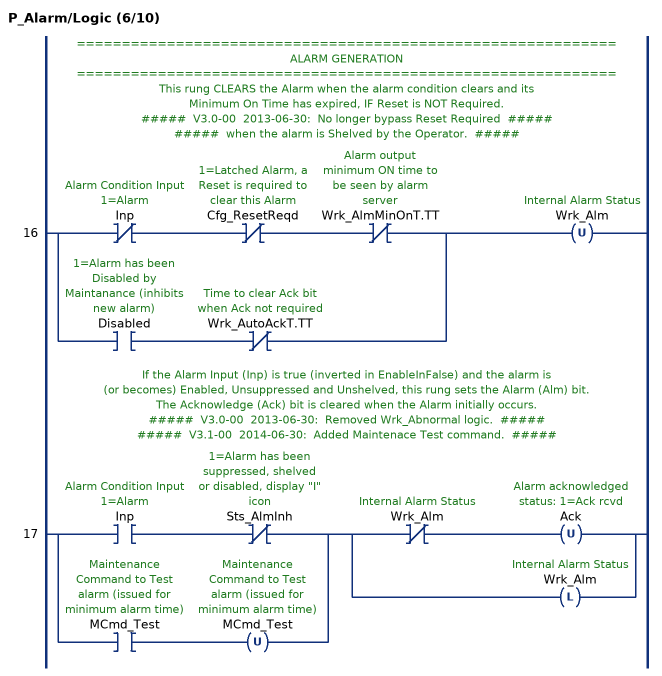
   // ============================================================
   // ALARM GENERATION
   // ============================================================
   // This rung CLEARS the Alarm when the alarm condition clears and its
   // Minimum On Time has expired, IF Reset is NOT Required.
   // #####  V3.0-00  2013-06-30:  No longer bypass Reset Required  #####
   // #####  when the alarm is Shelved by the Operator.  #####
   16: [XIO(Inp) XIO(Cfg_ResetReqd) XIO(Wrk_AlmMinOnT.TT) ,XIC(Disabled) XIO(Wrk_AutoAckT.TT) ]OTU(Wrk_Alm);
   // If the Alarm Input (Inp) is true (inverted in EnableInFalse) and the alarm is
   // (or becomes) Enabled, Unsuppressed and Unshelved, this rung sets the Alarm (Alm) bit.
   // The Acknowledge (Ack) bit is cleared when the Alarm initially occurs.
   // #####  V3.0-00  2013-06-30:  Removed Wrk_Abnormal logic.  #####
   // #####  V3.1-00  2014-06-30:  Added Maintenace Test command.  #####
   17: [XIC(Inp) XIO(Sts_AlmInh) ,XIC(MCmd_Test) OTU(MCmd_Test) ][XIO(Wrk_Alm) OTU(Ack) ,OTL(Wrk_Alm) ];
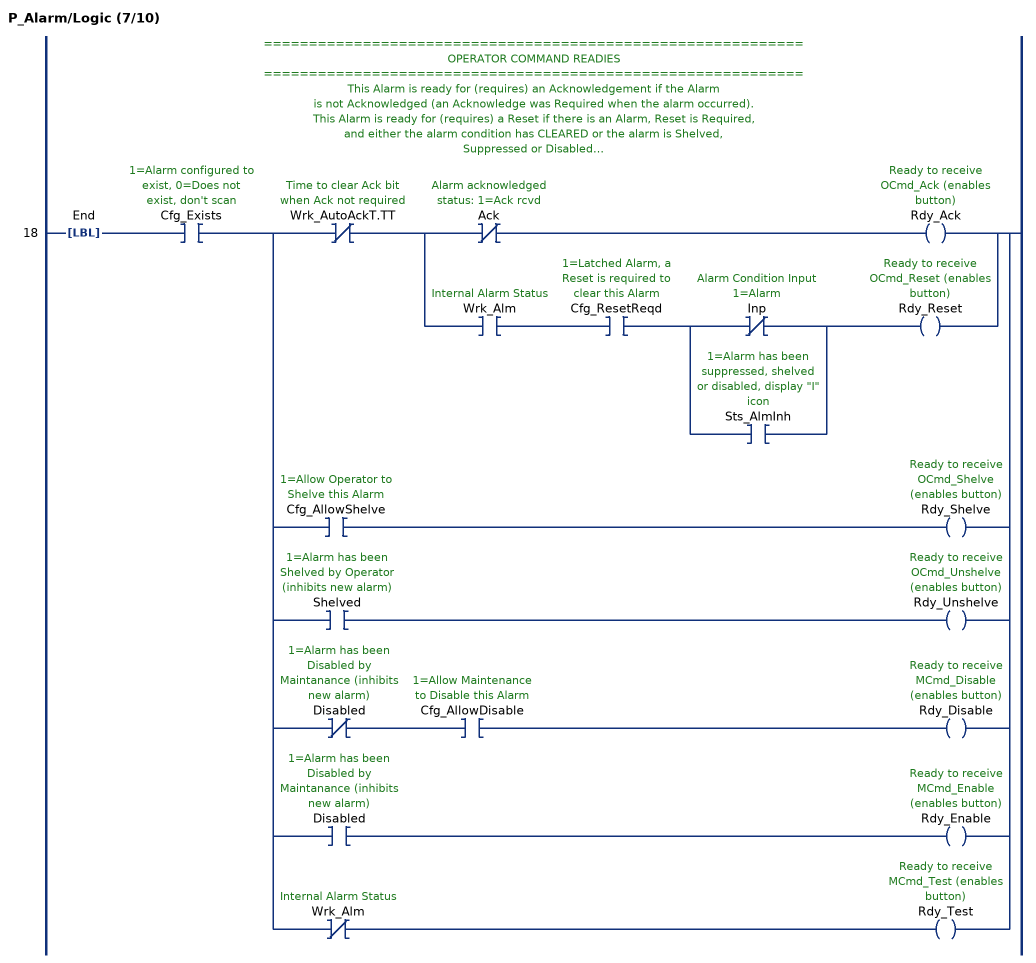
   // ============================================================
   // OPERATOR COMMAND READIES
   // ============================================================
   // This Alarm is ready for (requires) an Acknowledgement if the Alarm
   // is not Acknowledged (an Acknowledge was Required when the alarm occurred).
   // This Alarm is ready for (requires) a Reset if there is an Alarm, Reset is Required,
   // and either the alarm condition has CLEARED or the alarm is Shelved,
   // Suppressed or Disabled.
   // .
   // If the Alarm is NOT Shelved, it is ready for Shelve.
   // If the Alarm IS Shelved, it is ready for Unshelve.
   // If the Alarm is NOT Disabled, it is ready for Disable.
   // If the Alarm IS Disabled, it is ready for Enable.
   // NOTE: This rung appears before the Values/Status rung because the Rdy_Reset
   // condition is used to eliminate redundant logic in the rung below for Val_Notify.0.
   // #####  V3.0-00  2013-06-30:  Added sub-branch with Sts_AlmInh  #####
   // #####  V3.1-00  2014-06-30:  Added Maintenace Test command.  #####
   18: LBL(End)XIC(Cfg_Exists)[XIO(Wrk_AutoAckT.TT) [XIO(Ack) OTE(Rdy_Ack) ,XIC(Wrk_Alm) XIC(Cfg_ResetReqd) [XIO(Inp) ,XIC(Sts_AlmInh) ] OTE(Rdy_Reset) ] ,XIC(Cfg_AllowShelve) OTE(Rdy_Shelve) ,XIC(Shelved) OTE(Rdy_Unshelve) ,XIO(Disabled) XIC(Cfg_AllowDisable) OTE(Rdy_Disable) ,XIC(Disabled) OTE(Rdy_Enable) ,XIO(Wrk_Alm) OTE(Rdy_Test) ];
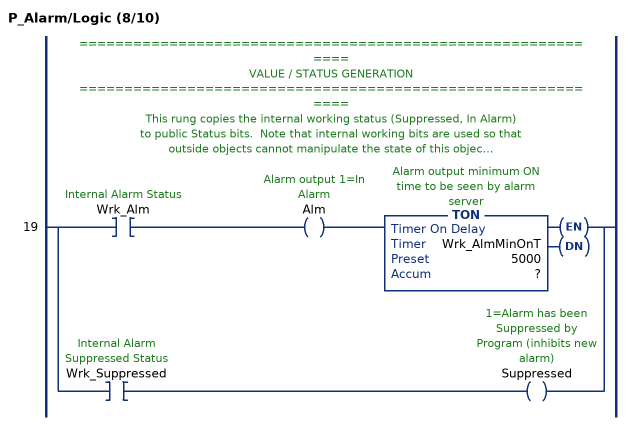
   // ============================================================
   // VALUE / STATUS GENERATION
   // ============================================================
   // This rung copies the internal working status (Suppressed, In Alarm)
   // to public Status bits.  Note that internal working bits are used so that
   // outside objects cannot manipulate the state of this object
   // by setting/clearing its Status and Alarm bits.
   // Public Status is generated for:
   // Alarm (with minimum ON time to be seen by polling)
   // Alarm Suppressed
   // Unsuppressed, Unshelved and Enabled are generated for HMI (FTVSE 7).
   // (Ack, Shelved and Disabled can be set/cleared by the HMI directly.
   // Note that these bits are "read/write" outputs in the parameter definition.)
   // #####  V3.0-00  2013-06-30:  New rung, some from below, new HMI bits.  #####
   19: [XIC(Wrk_Alm) OTE(Alm) TON(Wrk_AlmMinOnT,?,?) ,XIC(Wrk_Suppressed) OTE(Suppressed) ];
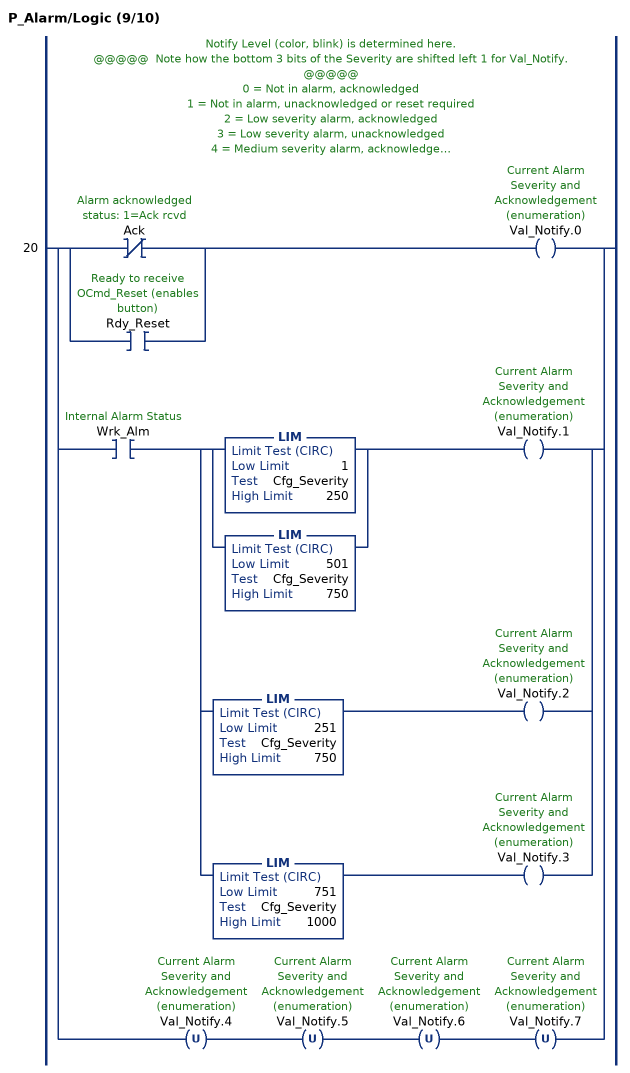
   // Notify Level (color, blink) is determined here.
   // @@@@@  Note how the bottom 3 bits of the Severity are shifted left 1 for Val_Notify.  @@@@@
   // 0 = Not in alarm, acknowledged
   // 1 = Not in alarm, unacknowledged or reset required
   // 2 = Low severity alarm, acknowledged
   // 3 = Low severity alarm, unacknowledged
   // 4 = Medium severity alarm, acknowledged
   // 5 = Medium severity alarm, unacknowledged
   // 6 = High severity alarm, acknowledged
   // 7 = High severity alarm, unacknowledged
   // 8 = Urgent severity alarm, acknowledged
   // 9 = Urgent severity alarm, unacknowledged
   // NOTE that the alarm bell icon will blink, even though the alarm is Acknowledged,
   // if an Alarm Reset is required (to get the Operator's attention).
   // #####  V3.0-00  2013-06-30:  Moved a few functions off this rung to logic above.  #####
   // #####  Names of Severity levels changed to Low, Medium, High, Highest  #####
   // #####  to match examples in ANSI/ISA-18.2-2009.  #####
   // #####  V3.1-00  2014-06-30:  Changed severity ranges, names to match FTAE  #####
   20: [[XIO(Ack) ,XIC(Rdy_Reset) ] OTE(Val_Notify.0) ,XIC(Wrk_Alm) [[LIM(1,Cfg_Severity,250) ,LIM(501,Cfg_Severity,750) ] OTE(Val_Notify.1) ,LIM(251,Cfg_Severity,750) OTE(Val_Notify.2) ,LIM(751,Cfg_Severity,1000) OTE(Val_Notify.3) ] ,OTU(Val_Notify.4) OTU(Val_Notify.5) OTU(Val_Notify.6) OTU(Val_Notify.7) ];
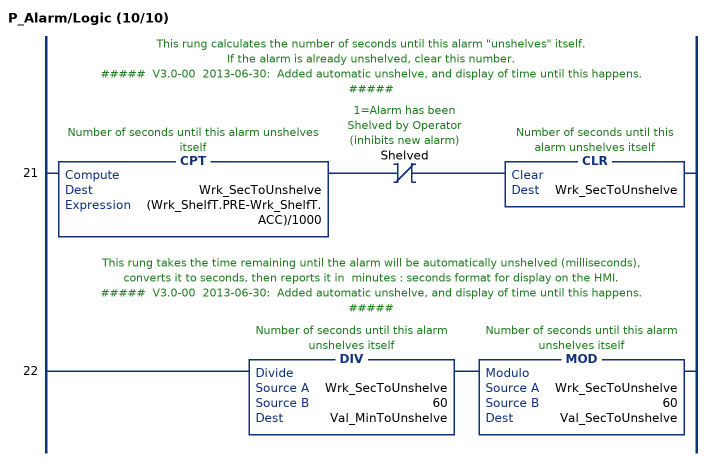
   // This rung calculates the number of seconds until this alarm "unshelves" itself.
   // If the alarm is already unshelved, clear this number.
   // #####  V3.0-00  2013-06-30:  Added automatic unshelve, and display of time until this happens.  #####
   21: CPT(Wrk_SecToUnshelve,(Wrk_ShelfT.PRE-Wrk_ShelfT.ACC)/1000)XIO(Shelved)CLR(Wrk_SecToUnshelve);
   // This rung takes the time remaining until the alarm will be automatically unshelved (milliseconds),
   // converts it to seconds, then reports it in  minutes : seconds format for display on the HMI.
   // #####  V3.0-00  2013-06-30:  Added automatic unshelve, and display of time until this happens.  #####
   22: DIV(Wrk_SecToUnshelve,60,Val_MinToUnshelve)MOD(Wrk_SecToUnshelve,60,Val_SecToUnshelve);
END_ROUTINE
